Yaskawa INFORM job: aruba_cylinder_program.JBI

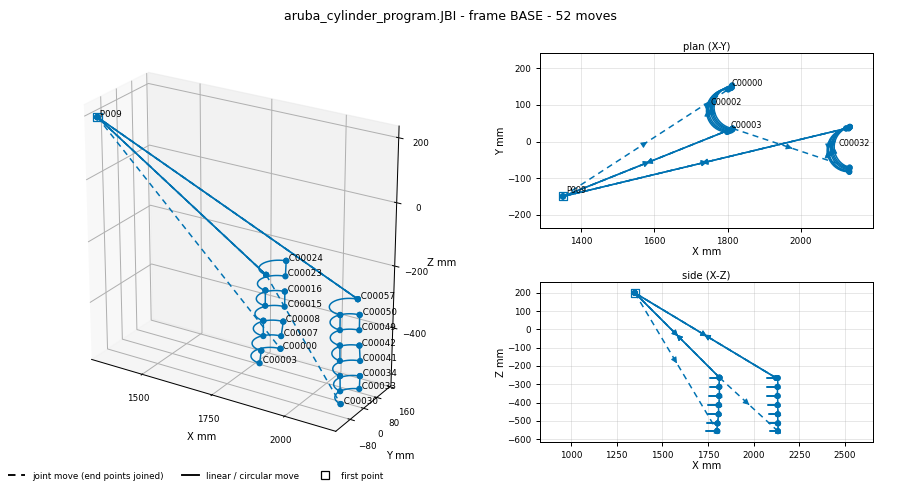
[picture p0: tool path of aruba_cylinder_program.JBI in frame BASE, 52 of 66 moves have a stored position in this frame; points joined in program order, loops and branches not executed]
/JOB
//NAME aruba_cylinder_program
//POS
///NPOS 60,0,60,1,0,1
///TOOL 0
///POSTYPE BASE
///RECTAN
///RCONF 0,0,0,0,0,0,0,0,0,0,0,0,0,0,0,0,0,0,0,0,0,0,0,0
C00000=1801.640,142.440,-556.605,-90.0000,-90.0000,5.0000
C00001=1801.640,142.440,-556.605,-90.0000,-90.0000,5.0000
C00002=1742.400,89.912,-556.605,0.0000,-89.9999,5.0000
C00003=1798.480,25.792,-556.605,90.0000,-90.0000,5.0000
C00004=1802.720,28.110,-514.228,90.0000,-90.0000,5.0000
C00005=1802.720,28.110,-514.228,90.0000,-90.0000,5.0000
C00006=1744.620,83.272,-514.228,0.0000,-89.9999,5.0000
C00007=1802.530,144.286,-514.228,-90.0000,-90.0000,5.0000
C00008=1808.630,145.913,-464.228,-90.0000,-90.0000,5.0000
C00009=1808.630,145.913,-464.228,-90.0000,-90.0000,5.0000
C00010=1747.980,84.019,-464.228,0.0000,-89.9999,5.0000
C00011=1808.740,29.691,-464.228,90.0000,-90.0000,5.0000
C00012=1807.810,31.178,-414.228,90.0000,-90.0000,5.0000
C00013=1807.810,31.178,-414.228,90.0000,-90.0000,5.0000
C00014=1752.660,86.966,-414.228,0.0000,-89.9999,5.0000
C00015=1811.890,147.733,-414.228,-90.0000,-90.0000,5.0000
C00016=1811.090,149.347,-364.228,-90.0000,-90.0000,5.0000
C00017=1811.090,149.347,-364.228,-90.0000,-90.0000,5.0000
C00018=1756.190,87.908,-364.228,0.0000,-89.9999,5.0000
C00019=1813.120,32.580,-364.228,90.0000,-90.0000,5.0000
C00020=1812.580,33.920,-314.228,90.0000,-90.0000,5.0000
C00021=1812.580,33.920,-314.228,90.0000,-90.0000,5.0000
C00022=1759.430,87.264,-314.228,0.0000,-89.9999,5.0000
C00023=1811.640,150.950,-314.228,-90.0000,-90.0000,5.0000
C00024=1812.440,153.409,-263.917,-90.0000,-90.0000,5.0000
C00025=1812.440,153.409,-263.917,-90.0000,-90.0000,5.0000
C00026=1762.940,92.020,-263.917,0.0000,-89.9999,5.0000
C00027=1813.830,35.728,-263.917,90.0000,-90.0000,5.0000
C00028=1813.830,35.728,-263.917,90.0000,-90.0000,5.0000
C00029=1813.830,35.728,-263.917,90.0000,-90.0000,5.0000
C00030=2133.610,-70.976,-557.001,90.0000,-90.0000,5.0000
C00031=2133.610,-70.976,-557.001,90.0000,-90.0000,5.0000
C00032=2091.520,-21.465,-557.001,5.0000,-89.9999,5.0000
C00033=2133.490,40.392,-557.001,-90.0000,-90.0000,5.0000
C00034=2134.550,40.359,-514.228,-90.0000,-90.0000,5.0000
C00035=2134.550,40.359,-514.228,-90.0000,-90.0000,5.0000
C00036=2087.100,-16.815,-514.228,5.0000,-89.9999,5.0000
C00037=2132.560,-73.356,-514.228,90.0000,-90.0000,5.0000
C00038=2132.220,-75.502,-464.228,90.0000,-90.0000,5.0000
C00039=2132.220,-75.502,-464.228,90.0000,-90.0000,5.0000
C00040=2084.190,-21.826,-464.228,5.0000,-89.9999,5.0000
C00041=2134.500,39.433,-464.228,-90.0000,-90.0000,5.0000
C00042=2131.580,38.031,-414.228,-90.0000,-90.0000,5.0000
C00043=2131.580,38.031,-414.228,-90.0000,-90.0000,5.0000
C00044=2080.940,-19.750,-414.228,5.0000,-89.9999,5.0000
C00045=2131.940,-77.487,-414.228,90.0000,-90.0000,5.0000
C00046=2132.030,-79.560,-364.228,90.0000,-90.0000,5.0000
C00047=2132.030,-79.560,-364.228,90.0000,-90.0000,5.0000
C00048=2075.660,-23.565,-364.228,5.0000,-89.9999,5.0000
C00049=2130.560,37.000,-364.228,-90.0000,-90.0000,5.0000
C00050=2131.060,36.010,-314.228,-90.0000,-90.0000,5.0000
C00051=2131.060,36.010,-314.228,-90.0000,-90.0000,5.0000
C00052=2074.880,-21.424,-314.228,5.0000,-89.9999,5.0000
C00053=2132.130,-81.339,-314.228,90.0000,-90.0000,5.0000
C00054=2132.550,-82.733,-265.632,90.0000,-90.0000,5.0000
C00055=2132.550,-82.733,-265.632,90.0000,-90.0000,5.0000
C00056=2072.250,-17.091,-265.632,5.0000,-89.9999,5.0000
C00057=2123.860,35.842,-265.632,-90.0000,-90.0000,5.0000
C00058=2123.860,35.842,-265.632,-90.0000,-90.0000,5.0000
C00059=2123.860,35.842,-265.632,-90.0000,-90.0000,5.0000
///POSTYPE PULSE
///PULSE
EC00000=0
EC00001=0
EC00002=0
EC00003=0
EC00004=0
EC00005=0
EC00006=0
EC00007=0
EC00008=0
EC00009=0
EC00010=0
EC00011=0
EC00012=0
EC00013=0
EC00014=0
EC00015=0
EC00016=0
EC00017=0
EC00018=0
EC00019=0
EC00020=0
EC00021=0
EC00022=0
EC00023=0
EC00024=0
EC00025=0
EC00026=0
EC00027=0
EC00028=0
EC00029=0
EC00030=0
EC00031=0
EC00032=0
EC00033=0
EC00034=0
EC00035=0
EC00036=0
EC00037=0
EC00038=0
EC00039=0
EC00040=0
EC00041=0
EC00042=0
EC00043=0
EC00044=0
EC00045=0
EC00046=0
EC00047=0
EC00048=0
EC00049=0
EC00050=0
EC00051=0
EC00052=0
EC00053=0
EC00054=0
EC00055=0
EC00056=0
EC00057=0
EC00058=0
EC00059=0
///POSTYPE BASE
///RECTAN
///RCONF 1,0,0,0,0,0,0,0,0,0,0,0,0,0,0,0,0,0,0,0,0,0,0,0
P00009=1350.000,-150.000,200.000,-180.0000,-45.0000,0.0000
///POSTYPE PULSE
///PULSE
EX00000=0
//INST
///DATE 2023/05/11 16:47
///ATTR SC,RW,RJ
////FRAME BASE
///GROUP1 RB1,ST1
NOP
MOVJ P009 EX000 VJ=15.00
MOVJ P009 VJ=15.00
MOVJ C00000 EC00000 VJ=15.00
MOVC C00001 EC00001 V=50.0
MOVC C00002 EC00002 V=50.0
MOVC C00003 EC00003 V=50.0
MOVL C00004 EC00004 V=50.0
MOVC C00005 EC00005 V=50.0
MOVC C00006 EC00006 V=50.0
MOVC C00007 EC00007 V=50.0
MOVL C00008 EC00008 V=50.0
MOVC C00009 EC00009 V=50.0
MOVC C00010 EC00010 V=50.0
MOVC C00011 EC00011 V=50.0
MOVL C00012 EC00012 V=50.0
MOVC C00013 EC00013 V=50.0
MOVC C00014 EC00014 V=50.0
MOVC C00015 EC00015 V=50.0
MOVL C00016 EC00016 V=50.0
MOVC C00017 EC00017 V=50.0
MOVC C00018 EC00018 V=50.0
MOVC C00019 EC00019 V=50.0
MOVL C00020 EC00020 V=50.0
MOVC C00021 EC00021 V=50.0
MOVC C00022 EC00022 V=50.0
MOVC C00023 EC00023 V=50.0
MOVL C00024 EC00024 V=50.0
MOVC C00025 EC00025 V=50.0
MOVC C00026 EC00026 V=50.0
MOVC C00027 EC00027 V=50.0
CALL JOB:SPYOF
MOVJ P009 VJ=15.00
MOVL C00028 EC00028 V=50.0
MOVJ P009 VJ=15.00
MOVL C00029 EC00029 V=50.0
MOVJ C00030 EC00030 VJ=15.00
MOVC C00031 EC00031 V=50.0
MOVC C00032 EC00032 V=50.0
MOVC C00033 EC00033 V=50.0
MOVL C00034 EC00034 V=50.0
MOVC C00035 EC00035 V=50.0
MOVC C00036 EC00036 V=50.0
MOVC C00037 EC00037 V=50.0
MOVL C00038 EC00038 V=50.0
MOVC C00039 EC00039 V=50.0
MOVC C00040 EC00040 V=50.0
MOVC C00041 EC00041 V=50.0
MOVL C00042 EC00042 V=50.0
MOVC C00043 EC00043 V=50.0
MOVC C00044 EC00044 V=50.0
MOVC C00045 EC00045 V=50.0
MOVL C00046 EC00046 V=50.0
MOVC C00047 EC00047 V=50.0
MOVC C00048 EC00048 V=50.0
MOVC C00049 EC00049 V=50.0
MOVL C00050 EC00050 V=50.0
MOVC C00051 EC00051 V=50.0
MOVC C00052 EC00052 V=50.0
MOVC C00053 EC00053 V=50.0
MOVL C00054 EC00054 V=50.0
MOVC C00055 EC00055 V=50.0
MOVC C00056 EC00056 V=50.0
MOVC C00057 EC00057 V=50.0
MOVJ P009 VJ=15.00
MOVL C00058 EC00058 V=50.0
MOVJ P009 VJ=15.00
MOVL C00059 EC00059 V=50.0
END
